FUNCTION_BLOCK Conveyor_S_Adp (* Composite Function Block Type *)
  (* Standard: 61499-2 *)
  (* Version 0.0, 4/23/2020, prana, nxtControl GmbH, template *)
  PACKAGE Main;
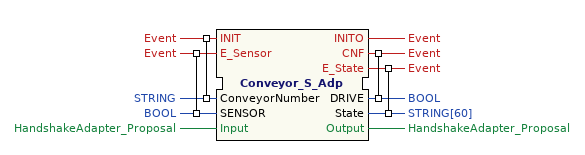
  EVENT_INPUT
    INIT WITH ConveyorNumber; (* Initialization Request *)
    E_Sensor WITH SENSOR;
  END_EVENT
  EVENT_OUTPUT
    INITO; (* Initialization Confirm *)
    CNF WITH DRIVE;
    E_State WITH State;
  END_EVENT
  VAR_INPUT
    ConveyorNumber : STRING;
    SENSOR : BOOL; (* Current value(i) in the named variable array element *)
  END_VAR
  VAR_OUTPUT
    DRIVE : BOOL;
    State : STRING[60];
  END_VAR
  SOCKETS
    Input : HandshakeAdapter_Proposal;
  END_SOCKETS
  PLUGS
    Output : HandshakeAdapter_Proposal;
  END_PLUGS
  FBS
    FB2 : StandardSection;
    FB3 : E_MERGE;
    ConveyorControl : ConveyorAdvanced;
    FB4 : OP_Select_Str;
    FB1 : E_SPLIT;
  END_FBS
  EVENT_CONNECTIONS
    INIT TO FB2.INIT;
    ConveyorControl.DRIVE_ON TO FB2.DRIVE_ON;
    ConveyorControl.DRIVE_OFF TO FB2.DRIVE_OFF;
    FB3.EO TO CNF;
    FB2.E_SENSOR TO FB3.EI2;
    ConveyorControl.DRIVE_ON TO FB3.EI1;
    ConveyorControl.DRIVE_OFF TO FB3.EI1;
    ConveyorControl.DONE TO FB4.Block1;
    ConveyorControl.E_CommandOut TO Output.E_Data1;
    Input.E_Data1 TO ConveyorControl.E_Command;
    E_Sensor TO Output.E_Data2;
    Input.E_Data2 TO ConveyorControl.E_PrevSensor;
    E_Sensor TO Input.E_Data5;
    Output.E_Data5 TO ConveyorControl.E_NextSensor;
    FB4.E_OP TO Input.E_Data4;
    Output.E_Data4 TO FB4.Block2;
    FB2.INITO TO INITO;
    ConveyorControl.E_State TO E_State;
    E_Sensor TO ConveyorControl.E_SensorCurrent;
    Input.E_Data3 TO FB1.EI;
    FB1.EO1 TO ConveyorControl.Reset;
    FB1.EO2 TO Output.E_Data3;
  END_CONNECTIONS
  DATA_CONNECTIONS
    ConveyorControl.DRIVE TO DRIVE;
    ConveyorNumber TO ConveyorControl.ConveyorNumber;
    ConveyorControl.OpConfirmation TO FB4.Data1;
    ConveyorControl.CommandOut TO Output.Data1;
    Input.Data1 TO ConveyorControl.Command;
    SENSOR TO Output.Data2;
    SENSOR TO Input.Data5;
    Output.Data5 TO ConveyorControl.NextSensor;
    FB4.Output TO Input.Data4;
    Output.Data4 TO FB4.Data2;
    Input.Data2 TO ConveyorControl.PrevSensor;
    ConveyorControl.State TO State;
    SENSOR TO ConveyorControl.CurrentSensor;
  END_CONNECTIONS
END_FUNCTION_BLOCK
